// TIA Portal V17 export
// export: Created 2025-03-13T10:30:57.1573106Z, ExportSetting WithDefaults, DisplayName Totally Integrated Automation Portal, DisplayVersion V17 Update 8, DisplayName TIA Portal Openness, DisplayVersion V17 Update 8, DisplayName TIA Portal Version Control Interface, DisplayVersion V17, DisplayName SINAMICS Startdrive Advanced, DisplayVersion V17 SP2, DisplayName SINAMICS Startdrive G110M, G120, G120C, G120D, G120P, G115D, DisplayVersion V17 SP2, DisplayName SINAMICS Startdrive G130, G150, S120, S150, SINAMICS MV, S210, DisplayVersion V17 SP2, DisplayName STEP 7 Professional, DisplayVersion V17 Update 8, DisplayName SINUMERIK ONE STEP 7 Toolbox, DisplayVersion V17 Update 12, DisplayName SINUMERIK 840D sl STEP 7 Toolbox, DisplayVersion V17 Update 12, DisplayName STEP 7 Safety, DisplayVersion V17 Update 6, DisplayName WinCC Advanced, DisplayVersion V17 Update 8
DATA_BLOCK "DB1463_CELL_COOLING_BUFFER_AUX_SYSTEM"   // DB1463
AUTHOR : ETXETAR
VERSION : 1.0
// stored: AutoNumber false, DBAccessibleFromOPCUA true, DBAccessibleFromWebserver true, InstanceOfName FB1452_AUXILIARY_COOLING_SYSTEM, InstanceOfType FB
"FB1452_AUXILIARY_COOLING_SYSTEM"
   // VAR_INPUT
   //    OPTIONS_0 : Byte;
   //    OPTIONS_1 : Byte;
   //    CIRCUIT_BREAKER_INPUT : Bool;
   //    CONTACTOR_FEEDBACK : Bool;
   //    LOW_LEVEL_ALM : Bool;
   //    OVERTEMPERATURE_ALM : Bool;
   //    U01_FLOW_ACTUAL_RAW_VALUE : Int;
   //    U01_TEMP_ACTUAL_RAW_VALUE : Int;
   //    U02_FLOW_ACTUAL_RAW_VALUE : Int;
   //    U02_TEMP_ACTUAL_RAW_VALUE : Int;
   //    HMI_REQ_LINE : Bool;
   // END_VAR
   // VAR_OUTPUT
   //    U01_U02_BREAKER_TRIPPED_ALARM : Bool;
   //    U01_U02_CONTACTOR_FEEDBACK_ALARM : Bool;
   //    U01_U02_LOW_LEVEL_INPUT_ALARM : Bool;
   //    U01_U02_OVERTEMPERATURE_INPUT_ALARM : Bool;
   //    U01_FLOW_FEEDBACK_ALARM : Bool;
   //    U01_FLOW_HIGH_LIMIT_ALARM : Bool;
   //    U01_FLOW_HIGH_LIMIT_WARNING : Bool;
   //    U01_FLOW_LOW_LIMIT_ALARM : Bool;
   //    U01_FLOW_LOW_LIMIT_WARNING : Bool;
   //    U01_TEMP_HIGH_LIMIT_ALARM : Bool;
   //    U01_TEMP_HIGH_LIMIT_WARNING : Bool;
   //    U01_TEMP_LOW_LIMIT_ALARM : Bool;
   //    U01_TEMP_LOW_LIMIT_WARNING : Bool;
   //    U01_FLOW_SETPOINT_ALARM : Bool;
   //    U01_TEMP_SETPOINT_ALARM : Bool;
   //    U02_FLOW_FEEDBACK_ALARM : Bool;
   //    U02_FLOW_HIGH_LIMIT_ALARM : Bool;
   //    U02_FLOW_HIGH_LIMIT_WARNING : Bool;
   //    U02_FLOW_LOW_LIMIT_ALARM : Bool;
   //    U02_FLOW_LOW_LIMIT_WARNING : Bool;
   //    U02_TEMP_HIGH_LIMIT_ALARM : Bool;
   //    U02_TEMP_HIGH_LIMIT_WARNING : Bool;
   //    U02_TEMP_LOW_LIMIT_ALARM : Bool;
   //    U02_TEMP_LOW_LIMIT_WARNING : Bool;
   //    U02_FLOW_SETPOINT_ALARM : Bool;
   //    U02_TEMP_SETPOINT_ALARM : Bool;
   //    HMI_POWER_UP_COND_OFF : Bool;
   //    HMI_POWER_UP_COND_ON : Bool;
   //    HMI_POWER_UP_EXECU_LEFT : Bool;
   //    HMI_POWER_UP_EXECU_RIGHT : Bool;
   //    MAIN_VALVE : Bool;
   // END_VAR
   // VAR
   //    SWITCH_ON_GENERAL_CONDITIONS : Bool;
   //    SWITCH_ON_INITIAL_CONDITIONS : Bool;
   //    SWITCH_ON_MANUAL_REQUEST : Bool;
   //    SWITCH_ON_AUTO_REQUEST : Bool;
   //    SWITCH_ON_GLOBAL_REQUEST : Bool;
   //    SWITCH_ON_COMMAND : Bool;
   //    SWITCH_ON : Bool;
   //    IN_SERVICE : Bool;
   //    SWITCH_OFF_GENERAL_CONDITIONS : Bool;
   //    SWITCH_OFF_INITIAL_CONDITIONS : Bool;
   //    SWITCH_OFF_MANUAL_REQUEST : Bool;
   //    SWITCH_OFF_AUTO_REQUEST : Bool;
   //    SWITCH_OFF_GLOBAL_REQUEST : Bool;
   //    SWITCH_OFF_COMMAND : Bool;
   //    SWITCH_OFF : Bool;
   //    OUT_OF_SERVICE : Bool;
   //    MANUAL_REQUEST_HELP : Bool;
   //    SWITCH_ON_GENERAL_CONDITION_HELP : Bool;
   //    SWITCH_ON_INITIAL_CONDITION_HELP : Bool;
   //    SWITCH_OFF_GENERAL_CONDITION_HELP : Bool;
   //    SWITCH_OFF_INITIAL_CONDITION_HELP : Bool;
   //    ANY_ACTIVE_ALARM : Bool;
   //    SEOC_ALARMS : Bool;
   //    WARNINGS : Bool;
   //    WARNINGS_GONE : Bool;
   //    UNIT_01_FLOW_FEEDBACK_INPUT : Bool;
   //    UNIT_02_FLOW_FEEDBACK_INPUT : Bool;
   //    TOTAL_FLOW_FEEDBACK_INPUT : Bool;
   //    AUX_COOLING_SENSOR_U01_VALUES { ExternalAccessible := 'False'; ExternalVisible := 'False'; ExternalWritable := 'False'} : "COOLING_SENSOR";
   //    AUX_COOLING_SENSOR_U02_VALUES { ExternalAccessible := 'False'; ExternalVisible := 'False'; ExternalWritable := 'False'} : "COOLING_SENSOR";
   //    TIMER_CONVEYOR_CONTACTOR_RELAY_ALARM : TON_TIME;
   // END_VAR
BEGIN
END_DATA_BLOCK
